Fanuc KAREL source: APPEND_NODE.kl

PROGRAM T
%NOLOCKGROUP
VAR
 v0 : PATH
 v1 : INTEGER
BEGIN
 APPEND_NODE(v0, v1)
END T
